KUKA KRL program: chk_w6_wechs_ok.src

&ACCESS RV5
&COMMENT Check Gripper Axor
DEF chk_w6_wechs_ok( )

; VERIFICAÇÃO DE FERRAMENTA: Gripper Axor

WAIT FOR ((($in [161]) AND ($in[169])) AND ($in[177]) AND ($in[185]) AND ($in[193]) AND (NOT $in[201]) AND ( $in[219]) AND NOT ($IN[3320]))

END
